FUNCTION_BLOCK ChanRcvBool (* Composite Function Block Type *)
  (* Standard: 61499-2 *)
  (* Version 0.0, 7/15/2023, vv263, nxtControl GmBH, template *)
  PACKAGE Main;
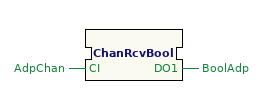
  SOCKETS
    CI : AdpChan;
  END_SOCKETS
  PLUGS
    DO1 : BoolAdp;
  END_PLUGS
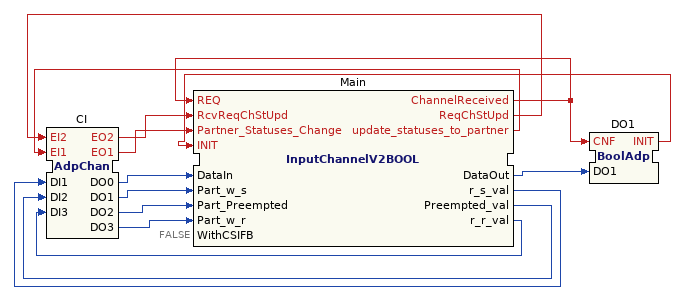
  FBS
    Main : InputChannelV2BOOL(WithCSIFB := FALSE);
  END_FBS
  EVENT_CONNECTIONS
    Main.ChannelReceived TO DO1.CNF;
    Main.ChannelReceived TO Main.REQ;
    CI.EO2 TO Main.RcvReqChStUpd;
    CI.EO1 TO Main.Partner_Statuses_Change;
    Main.ReqChStUpd TO CI.EI2;
    Main.update_statuses_to_partner TO CI.EI1;
    DO1.INIT TO Main.INIT;
  END_CONNECTIONS
  DATA_CONNECTIONS
    Main.DataOut TO DO1.DO1;
    CI.DO0 TO Main.DataIn;
    CI.DO1 TO Main.Part_w_s;
    CI.DO2 TO Main.Part_Preempted;
    CI.DO3 TO Main.Part_w_r;
    Main.r_s_val TO CI.DI1;
    Main.Preempted_val TO CI.DI2;
    Main.r_r_val TO CI.DI3;
  END_CONNECTIONS
END_FUNCTION_BLOCK
